// TIA Portal project "学习上升沿下降沿" (V15.1)

(* hardware
DEVICE "S7-1200 station_1"  S7-1200 Station
   slot 0: "Rack_0"  S7-1200 Rack  Rack  V1.0
   slot 1: "PLC_1"  CPU 1212C DC/DC/DC  6ES7 212-1AE40-0XB0  V4.2
*)

// ===== PLC "PLC_1"  CPU 1212C DC/DC/DC =====

VAR_GLOBAL   // PLC tag table "默认变量表"
   ""上升"" AT %I0.0 : Bool;
   ""下降"" AT %I0.1 : Bool;
   ""上升1"" AT %I0.2 : Bool;
   ""下降1"" AT %I0.3 : Bool;
   ""总开关"" AT %I0.4 : Bool;
   ""保护开关"" AT %I0.5 : Bool;
   ""输出"" AT %Q0.0 : Bool;
   ""输出(1)"" AT %Q0.1 : Bool;
END_VAR